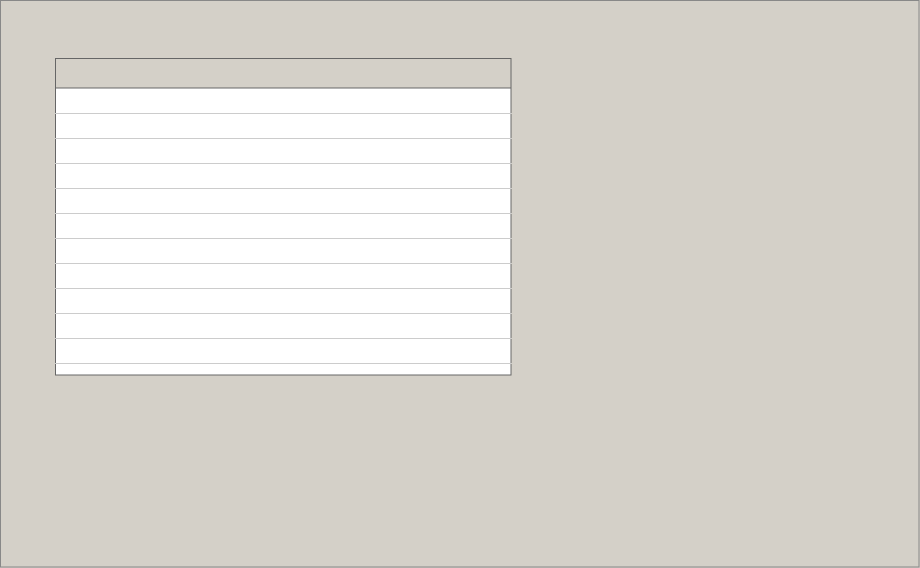
VISUALIZATION Model  // 920x568
AR_IN_OUT
	
END_VAR
    Table (55,58 456x317), data array: astModel
        p2170511999: astModel[INDEX].arPosition
        p3723444502: astModel[INDEX].arSpeed
        p1014161805: (GVL_RETAIN.cMaxModelNo - 1) - 0 + INT#1
        p1755163831: Type
        p1791247317: astModel[INDEX].abType
        p511219082: type
        p3312258591: astModel[INDEX].aiType
        p2232123230: Name
        p2685023577: astModel[INDEX].sName
END_VISUALIZATION

(* stored: Version 1.1.0.1
   Visu Model: Id {1ad760d6-49f5-452c-b8f8-8c412b5e472d} *)
